(*
SPDX-FileCopyrightText: © 2026 Oleksandr Tiutyk <trofimich@gmail.com>
SPDX-License-Identifier: MIT
License: https://opensource.org/license/mit
*)

(*!
<summary>Demonstrates construction and cyclic execution of a workflow.</summary>
<description>
Dynamically created activities and conditions are explicitly registered immediately after allocation checks,
before configuration.
</description>
*)

{attribute 'no_explicit_call' := 'do not call this function block directly'}
FUNCTION_BLOCK DemoWorkflowController EXTENDS TOF_Automation.AutomationController<0>
VAR
	_ElementFactory : DemoWorkflowElementFactory;
END_VAR
VAR_OUTPUT
	DemoWorkflow : DemoWorkflow;	
END_VAR
VAR_STAT	
	{attribute 'hide'} 
	_ClassName : STRING := __POUNAME();
END_VAR

(*!
<summary>Constructs workflow activities and transfers their ownership before configuration.</summary>
<description>
Creates owned elements through the common factory path. Later configuration failures leave
registered elements owned by the workflow for disposal.
</description>
<param name="workflow">Owner workflow instance.</param>
<param name="parentSequence">Parent sequence to append the activities to.</param>
<param name="cornerNumber">One-based corner index (1..4).</param>
*)
METHOD PRIVATE addMoveFromToActivity 
VAR_INPUT
	workflow : TOF_Workflow.IWorkflow;
	parentSequence : TOF_Workflow.ISequenceActivity;
	cornerNumber : BYTE;
END_VAR
VAR
	element : TOF_Workflow.IWorkflowElement;
	trueValue : BOOL := TRUE;
	
	needMoveVariableName : STRING;	
	targetXPosition : INT;
	targetYPosition : INT;
	
	waitButtonPressActivity : TOF_Workflow.IWaitVariableValueActivity;
	moveActivity : IMoveFromToActivity;
END_VAR
// calculate variable values depending of current position (corner number 1-4)
CASE cornerNumber OF 
	1:
		needMoveVariableName := 'MoveFrom1To2';
		targetXPosition := 400;
		targetYPosition := 0;
		
	2:
		needMoveVariableName := 'MoveFrom2To3';
		targetXPosition := 400;
		targetYPosition := 300;
		
	3:
		needMoveVariableName := 'MoveFrom3To4';
		targetXPosition := 0;
		targetYPosition := 300;
		
	4:
		needMoveVariableName := 'MoveFrom4To1';
		targetXPosition := 0;
		targetYPosition := 0;
END_CASE

element := TOF_Workflow.Workflows.CreateElement(
	typeName := 'TOF_Workflow.WaitVariableValueActivity',
	workflow := workflow
);

requireElementInterface(
	found := __QUERYINTERFACE(element, waitButtonPressActivity),
	interfaceName := 'TOF_Workflow.IWaitVariableValueActivity'
);

waitButtonPressActivity.Name := TOF_Core.WideStrings.Concat255("Wait", TO_WSTRING(needMoveVariableName), "Activity");
waitButtonPressActivity.Configure(monitoredVariableName := needMoveVariableName, referenceValue := trueValue);

parentSequence.AddChildActivity(activity := waitButtonPressActivity);

element := TOF_Workflow.Workflows.CreateElement(
	typeName := TOF_Core.Strings.Concat255(CurrentNamespace.Name, '.MoveFromToActivity'),
	workflow := workflow,
	factory := _ElementFactory
);

requireElementInterface(
	found := __QUERYINTERFACE(element, moveActivity),
	interfaceName := 'IMoveFromToActivity'
);

moveActivity.Name := TOF_Core.WideStrings.Concat255(TO_WSTRING(needMoveVariableName), "Activity");
moveActivity.Configure(toXPosition := targetXPosition, toYPosition := targetYPosition);

parentSequence.AddChildActivity(activity := moveActivity);
END_METHOD

(*!
<summary>Gets the child automation components array reference (none for this controller).</summary>
*)
PROPERTY Children : REFERENCE TO ARRAY [0.._ChildCount - 1] OF TOF_Automation.IChildAutomationComponent
GET
Children REF= 0;
END_GET
END_PROPERTY

(*!
<summary>Gets the runtime class name of this object.</summary>
*)
{attribute 'monitoring' := 'call'}
PROPERTY ClassName : REFERENCE TO STRING
GET
ClassName REF= _ClassName;
END_GET
END_PROPERTY

(*!
<summary>Gets the namespace name of this object.</summary>
*)
{attribute 'monitoring' := 'call'}
PROPERTY NamespaceName : REFERENCE TO STRING
GET
NamespaceName REF= CurrentNamespace.Name;
END_GET
END_PROPERTY

(*!
<summary>Constructs workflow activities and transfers their ownership before configuration.</summary>
<description>
Creates owned elements through the common factory path. Later configuration failures leave
registered elements owned by the workflow for disposal.
</description>
*)
METHOD PROTECTED OnBeforeChildrenInitializing
VAR
	element : TOF_Workflow.IWorkflowElement;
	whileActivity : TOF_Workflow.IWhileActivity;
	loopSequence : TOF_Workflow.ISequenceActivity;
	trueCondition : TOF_Workflow.ITrueCondition;
END_VAR
element := TOF_Workflow.Workflows.CreateElement(
	typeName := 'TOF_Workflow.WhileActivity',
	workflow := DemoWorkflow
);

requireElementInterface(
	found := __QUERYINTERFACE(element, whileActivity),
	interfaceName := 'TOF_Workflow.IWhileActivity'
);

element := TOF_Workflow.Workflows.CreateElement(
	typeName := 'TOF_Workflow.SequenceActivity',
	workflow := DemoWorkflow
);

requireElementInterface(
	found := __QUERYINTERFACE(element, loopSequence),
	interfaceName := 'TOF_Workflow.ISequenceActivity'
);

element := TOF_Workflow.Workflows.CreateElement(
	typeName := 'TOF_Workflow.TrueCondition',
	workflow := DemoWorkflow
);

requireElementInterface(
	found := __QUERYINTERFACE(element, trueCondition),
	interfaceName := 'TOF_Workflow.ITrueCondition'
);

whileActivity.Configure(condition := trueCondition, body := loopSequence);

addMoveFromToActivity(workflow := DemoWorkflow, parentSequence := loopSequence, cornerNumber := 1);
addMoveFromToActivity(workflow := DemoWorkflow, parentSequence := loopSequence, cornerNumber := 2);
addMoveFromToActivity(workflow := DemoWorkflow, parentSequence := loopSequence, cornerNumber := 3);
addMoveFromToActivity(workflow := DemoWorkflow, parentSequence := loopSequence, cornerNumber := 4);

DemoWorkflow.SetRootActivity(rootActivity := whileActivity);
END_METHOD

(*!
<summary>Requests resetting of DemoWorkflow when the controller is reset.</summary>
*)
METHOD PROTECTED OnBeforeChildrenReset
IF DemoWorkflow.ResettingAllowed THEN
	DemoWorkflow.RequestReset();
END_IF
END_METHOD

(*!
<summary>Cancels DemoWorkflow when the controller stops and advances it until cancellation completes.</summary>
*)
METHOD PROTECTED OnBeforeChildrenStopped
IF DemoWorkflow.CancellingAllowed THEN
	DemoWorkflow.RequestCancel(reason := "External stop");
END_IF

IF DemoWorkflow.Busy THEN
	DemoWorkflow.Execute();
END_IF
END_METHOD

(*!
<summary>Starts DemoWorkflow on the first working cycle and executes it cyclically thereafter.</summary>
*)
METHOD PROTECTED OnBeforeChildrenWorking
VAR_INST
	started : BOOL;
END_VAR
IF started THEN
	DemoWorkflow.Execute();
ELSE
	DemoWorkflow.RequestStart();
	
	started := TRUE;
END_IF
END_METHOD

(*!
<summary>Gets the string representation of the current controller operational state.</summary>
*)
{attribute 'monitoring' := 'call'}
PROPERTY OperationalStateName : STRING(16)
GET
OperationalStateName := TO_STRING(_OperationalState);
END_GET
END_PROPERTY

(*!
<summary>Gets the size in bytes of this function block instance.</summary>
*)
{attribute 'monitoring' := 'call'}
PROPERTY SelfSize : ULINT
GET
SelfSize := XSIZEOF(THIS^);
END_GET
END_PROPERTY

(*!
<summary>Checks the configuration interface requested for a factory-created sample node.</summary>
<description>A failed query raises before the caller uses the result. The workflow retains the registered node.</description>
<param name="found">Result of the interface query.</param>
<param name="interfaceName">Expected configuration interface for diagnostics.</param>
*)
METHOD PRIVATE requireElementInterface
VAR_INPUT
	found : BOOL;
	interfaceName : STRING;
END_VAR
VAR
	message : TOF_Core.ERROR_MESSAGE;
END_VAR
IF found THEN
	RETURN;
END_IF

message := TOF_Core.WideStrings.Concat255("Created workflow element requires interface ", TO_WSTRING(interfaceName));
TOF_Workflow.WorkflowExceptions.ThrowWorkflowConfiguration(
	sourceNamespaceName := NamespaceName,
	sourceClassName := ClassName,
	sourcePOUName := __POUNAME(),
	sourcePosition := __POSITION(),
	message := message
);
END_METHOD

END_FUNCTION_BLOCK

(* stored: Version 1.1.0.1
   POU DemoWorkflowController: Id {dc096c7a-49dd-4129-a1d0-54dcfc137d76}, SpecialFunc None
   Folder Overriden members: Id {dec9ed42-9850-4632-8368-9c2c6d0a2bdb}
   Folder Service methods: Id {1828c457-8a78-48a2-9b87-64cb67bc8882}
   Method addMoveFromToActivity: Id {5aa5ff3a-92c3-4d8d-9a23-b811cd230c9d}
   Property Children: Id {8735154c-178f-4bcc-a2c4-80749379f15d}
   Get Get: Id {e2436b7e-47bc-4e03-b117-577110a01efc}
   Property ClassName: Id {ad6b5264-2d84-464d-8021-1d07f9d49884}
   Get Get: Id {897a4b58-f1c6-4661-8c68-f7b7183bfc21}
   Property NamespaceName: Id {938e57da-e42b-4b88-8eda-dae4a4febad2}
   Get Get: Id {5a6e3df0-fc18-48c5-84f1-c69b86c3fddd}
   Method OnBeforeChildrenInitializing: Id {76f3f662-77f5-4af2-be03-b0557314d068}
   Method OnBeforeChildrenReset: Id {c84e19b2-7a35-4d91-b620-9e4f1a8c2d73}
   Method OnBeforeChildrenStopped: Id {3c199eb9-4006-4b9a-98cf-6e3625336148}
   Method OnBeforeChildrenWorking: Id {2d7b684e-2908-4409-82de-f87452b1d410}
   Property OperationalStateName: Id {a420c5dc-2bb8-4e16-9768-680503fa8551}
   Get Get: Id {5cb6bc34-a729-4d81-bb44-8fd2db6da917}
   Property SelfSize: Id {e4928d85-ffb2-44cd-81d8-5da5452d15ff}
   Get Get: Id {f290be1b-b375-45a7-a2dc-21a7680125fb}
   Method requireElementInterface: Id {9dadd88b-1193-4169-8e64-e0f75ed97dbe} *)
